FUNCTION_BLOCK FB_PlanarXtsMover

VAR_INPUT
	nMoverId			    	: UDINT;
	iTcIoXtsXpuMover			: REFERENCE TO Tc3_XTS_Utility.I_TcIoXtsXpuMover;
	refTrackConfig				: REFERENCE TO ST_TrackConfig;
END_VAR

VAR
	_McPlanarMover				: Tc3_Mc3PlanarMotion.MC_PlanarMover;
	_PlanarTrail    			: Tc3_Mc3PlanarMotion.MC_PlanarTrackTrail;

	stXtsPositionInfo			: Tc3_XTS_Utility.ST_PositionInfo;
	
	MoverPhysics				: Tc3_Physics.PositionXYC;

	Mover				        : MoverSort;
	
	stMoverStatus				: ST_MoverStatus;
END_VAR

METHOD PROTECTED _M_IsOnSection : BOOL
VAR_INPUT
	XtsTrackId			: OTCID;
	SectorStartPosn		: LREAL;
	SectorEndPosn		: LREAL;
END_VAR
_M_IsOnSection	:= (stXtsPositionInfo.nTrackObjectid = XtsTrackId) AND
					IsBetween(value := stXtsPositionInfo.fTrackPosition, minV := SectorStartPosn, maxV := SectorEndPosn);
END_METHOD

METHOD PROTECTED _M_UpdateStatus
stMoverStatus.MoverInShortcut := 
	_M_IsOnSection(XtsTrackId := GVL_General.XtsOutterLoopOid, 
					SectorStartPosn := refTrackConfig.stTrackShortcutConfig.stTrackSectorConfig.SectorStartPosn, 
					SectorEndPosn := refTrackConfig.stTrackShortcutConfig.stTrackSectorConfig.SectorEndPosn);
END_METHOD

PROPERTY IsCommandedInShortcut : BOOL
GET
VAR
	nCounter: UDINT := 0;
END_VAR
_mcPlanarMover.GetTrackTrailInformation(_PlanarTrail);

IF _PlanarTrail.Error OR _PlanarTrail.Size < 1 THEN
   IsCommandedInShortcut := FALSE;
   RETURN;
END_IF
   
FOR nCounter := 0 TO _PlanarTrail.Size - 1 DO
	IF _PlanarTrail.GetTrackOidAt(nCounter) = GVL_Mc3.MC_Tracks[E_TrackNum.Small].MCTOPLC_STD.TrackOID  THEN
		IsCommandedInShortcut := TRUE;
		RETURN;
	END_IF
END_FOR

IsCommandedInShortcut := FALSE;
END_GET
END_PROPERTY

METHOD JoinTrack

VAR_INPUT
	feedback: REFERENCE TO MC_PlanarFeedback;
END_VAR

VAR_IN_OUT
	track: MC_PlanarTrack;
END_VAR
_McPlanarMover.JoinTrack(feedback, track, 0, 0);
END_METHOD

PROPERTY McPlanarMover : REFERENCE TO MC_PlanarMover
GET
McPlanarMover REF= _McPlanarMover;
END_GET
END_PROPERTY

PROPERTY P_MoverPhysics : REFERENCE TO Tc3_Physics.PositionXYC
GET
P_MoverPhysics	REF= MoverPhysics;
END_GET
END_PROPERTY

PROPERTY P_MoverStatus : REFERENCE TO ST_MoverStatus
GET
P_MoverStatus REF= stMoverStatus;
END_GET
END_PROPERTY

PROPERTY P_XPlanarMover : REFERENCE TO MoverSort
GET
P_XPlanarMover	REF= Mover;
END_GET
END_PROPERTY

PROPERTY P_XtsPositionInfo : REFERENCE TO Tc3_XTS_Utility.ST_PositionInfo
GET
P_XtsPositionInfo	REF= stXtsPositionInfo;
END_GET
END_PROPERTY

METHOD Update : PVOID
IF iTcIoXtsXpuMover <> Tc3_Module.NULL THEN
  stXtsPositionInfo	:= iTcIoXtsXpuMover.GetPositionInfo();
END_IF

_mcPlanarMover.Update();

_mcPlanarMover.GetTrackTrailInformation(_PlanarTrail);

Mover.MoverNumber 	:= nMoverId;
Mover.MoverPos    	:= _McPlanarMover.MCTOPLC.SETONTRACK.SetPos;
Mover.TrackID     	:= _McPlanarMover.MCTOPLC.SETONTRACK.TrackOID;
//MoverPhysics		:= 

{warning <'Method Not Called'>}
//_M_UpdateStatus();

IF _PlanarTrail.Error OR _PlanarTrail.Size <= 1 THEN
   RETURN;
END_IF

IF iTcIoXtsXpuMover <> Tc3_Module.NULL THEN
  //SmallCircle
  IF _PlanarTrail.GetTrackOidAt(1) = MC_Tracks[E_TrackNum.Small].MCTOPLC_STD.TrackOID   THEN
    iTcIoXtsXpuMover.SetActiveTrackObjectId(XtsShortcutOid);
  //BigCircle
  ELSIF _PlanarTrail.GetTrackOidAt(1) =MC_Tracks[E_TrackNum.Big].MCTOPLC_STD.TrackOID THEN
    iTcIoXtsXpuMover.SetActiveTrackObjectId(XtsOutterLoopOid);
  END_IF
END_IF
END_METHOD

END_FUNCTION_BLOCK

(* stored: Version 1.1.0.1
   POU FB_PlanarXtsMover: Id {e98e5f10-cdde-43fc-96da-1ae5f511366a}, SpecialFunc None
   Folder Methods: Id {497e6300-3e6d-49b8-a318-13b94b960f56}
   Folder Properties: Id {bafe569f-b5f0-4de9-ae48-854cd11ccd2e}
   Method _M_IsOnSection: Id {6fb38ca4-6b76-0afd-297f-a5f43cfa3834}
   Method _M_UpdateStatus: Id {5fb917e1-5646-02f6-26ca-dbbb331704b2}
   Property IsCommandedInShortcut: Id {e5e69e7e-f163-4728-82da-b10e582ce622}
   Get Get: Id {7a71ba46-249d-415a-b1f4-f1c52c07bed0}
   Method JoinTrack: Id {fd819ce6-c064-4bae-aa84-926325f13c12}
   Property McPlanarMover: Id {79d72b75-52b9-47c8-886e-5e60276bf5f1}
   Get Get: Id {71cad725-c4c4-49c5-9410-cee17b681f5a}
   Property P_MoverPhysics: Id {056b1259-392a-0821-097b-b08bee10a569}
   Get Get: Id {e7ba31e5-6730-0d69-35c1-51b7d57fd5fd}
   Property P_MoverStatus: Id {4597e151-4034-0716-26cd-3b84c52a00ed}
   Get Get: Id {c9b03fbe-77df-00fa-3e75-da43ee6790b6}
   Property P_XPlanarMover: Id {a5ac8d37-9108-0740-305c-d3b342270158}
   Get Get: Id {bae1975d-f945-0652-3748-976b73c4f7d6}
   Property P_XtsPositionInfo: Id {eee46ce5-009e-038a-12e5-cdbf8f2886af}
   Get Get: Id {58ff9574-093b-05dd-3592-27328f83735e}
   Method Update: Id {2a189ea7-97f2-4dc0-980a-fdde9c091766} *)
